FUNCTION_BLOCK FloorCarElevator (* Basic Function Block Type *)
  (* Standard: 61499-2 *)
  (* Version 0.0, 6/17/2016, Andrei, nxtControl GmbH, Template *)
  PACKAGE Main;
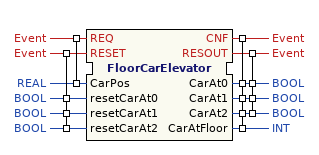
  EVENT_INPUT
    REQ WITH CarPos; (* Normal Execution Request *)
    RESET WITH resetCarAt0, resetCarAt1, resetCarAt2;
  END_EVENT
  EVENT_OUTPUT
    CNF WITH CarAt0, CarAt1, CarAt2, CarAtFloor; (* Execution Confirmation *)
    RESOUT WITH CarAt0, CarAt1, CarAt2;
  END_EVENT
  VAR_INPUT
    CarPos : REAL; (* Input event qualifier *)
    resetCarAt0 : BOOL;
    resetCarAt1 : BOOL;
    resetCarAt2 : BOOL;
  END_VAR
  VAR_OUTPUT
    CarAt0 : BOOL; (* Output event qualifier *)
    CarAt1 : BOOL;
    CarAt2 : BOOL;
    CarAtFloor : INT;
  END_VAR
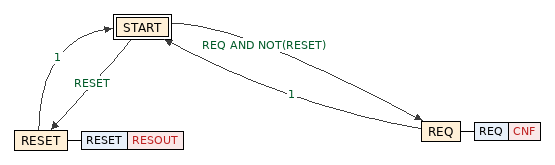
  EC_STATES
    START; (* Initial State *)
    REQ : REQ -> CNF; (* Normal execution *)
    RESET : RESET -> RESOUT;
  END_STATES
  EC_TRANSITIONS
    START TO REQ := REQ AND NOT(RESET);
    REQ TO START := 1;
    START TO RESET := RESET;
    RESET TO START := 1;
  END_TRANSITIONS
  ALGORITHM REQ IN ST: (* Normally executed algorithm *)
// Determine floor number of elevator
IF CarPos < 30.5 THEN
	CarAtFloor := 2;
	CarAt2 := TRUE;
	CarAt0 := FALSE;
	CarAt1 := FALSE;
ELSIF (CarPos  > 224.5) AND (CarPos < 225.5) THEN
	CarAtFloor := 1;
	CarAt1 := TRUE;
	CarAt0 := FALSE;
	CarAt2 := FALSE;
ELSIF CarPos > 418.5 THEN
	CarAtFloor := 0;
	CarAt0 := TRUE;
	CarAt1 := FALSE;
	CarAt2 := FALSE;
ELSE
	CarAt2 := FALSE;
	CarAt0 := FALSE;
	CarAt1 := FALSE;
END_IF;
  END_ALGORITHM
  ALGORITHM RESET IN ST:
CarAt0 := resetCarAt0;
CarAt1 := resetCarAt1;
CarAt2 := resetCarAt2;
IF (CarAt0) THEN
	CarAtFloor := 0;
ELSIF (CarAt1) THEN
	CarAtFloor := 1;
ELSIF CarAt2 THEN
	CarAtFloor := 2;
END_IF;
  END_ALGORITHM
END_FUNCTION_BLOCK
